KUKA KRL program: Milling_7_33.src

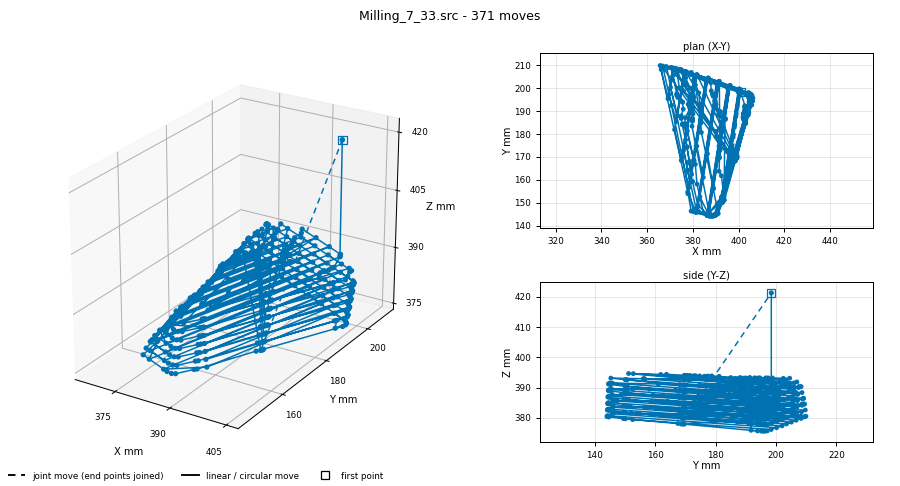
[picture p0: tool path of Milling_7_33.src, 371 of 373 moves have a stored position in this frame; points joined in program order, loops and branches not executed]
&ACCESS RVP
&REL 1
&PARAM TEMPLATE = C:\KRC\Roboter\Template\vorgabe
&PARAM EDITMASK = *
DEF Milling_7_33 ( )


;FOLD INI
;FOLD BASISTECH INI
GLOBAL INTERRUPT DECL 3 WHEN $STOPMESS==TRUE DO IR_STOPM ( )
INTERRUPT ON 3
BAS (#INITMOV,0 )
;ENDFOLD (BASISTECH INI)
;ENDFOLD (INI)

;FOLD STARTPOSITION - BASE IS 0, TOOL IS 5, SPEED IS 15%, POSITION IS A1 5,A2 -90,A3 100,A4 5,A5 -10,A6 -5,E1 0,E2 0,E3 0,E4 0
$BWDSTART = FALSE
PDAT_ACT = {VEL 15,ACC 100,APO_DIST 50}
FDAT_ACT = {TOOL_NO 5,BASE_NO 0,IPO_FRAME #BASE}
BAS (#PTP_PARAMS,15)
PTP  {A1 5,A2 -90,A3 100,A4 5,A5 -10,A6 -5,E1 0,E2 0,E3 0,E4 0}
;ENDFOLD

;FOLD LIN SPEED IS 0.1 m/sec, INTERPOLATION SETTINGS IN FOLD
$VEL.CP=0.1
$ADVANCE=3
;ENDFOLD

BAS(#VEL_PTP,2)
PTP {X 400.878, Y 198.448, Z 421.334, A -161.652, B 81.275, C -141.67, E1 0, E2 0, E3 0, E4 0, S 'B010'}
$VEL.CP=0.012
LIN {X 400.878, Y 198.448, Z 391.334, A -161.652, B 81.275, C -141.67, E1 0, E2 0, E3 0, E4 0}
LIN {X 393.619, Y 152.751, Z 394.599, A -161.652, B 81.275, C -141.67, E1 0, E2 0, E3 0, E4 0}
LIN {X 394.006, Y 186.825, Z 392.897, A -161.652, B 81.275, C -141.67, E1 0, E2 0, E3 0, E4 0}
LIN {X 396.301, Y 201.276, Z 391.864, A -161.652, B 81.275, C -141.67, E1 0, E2 0, E3 0, E4 0}
LIN {X 393.921, Y 186.294, Z 392.935, A -161.652, B 81.275, C -141.67, E1 0, E2 0, E3 0, E4 0}
LIN {X 391.87, Y 173.383, Z 393.857, A -161.652, B 81.275, C -141.67, E1 0, E2 0, E3 0, E4 0}
LIN {X 391.404, Y 170.446, Z 394.067, A -161.652, B 81.275, C -141.67, E1 0, E2 0, E3 0, E4 0}
LIN {X 391.763, Y 172.709, Z 393.905, A -161.652, B 81.275, C -141.67, E1 0, E2 0, E3 0, E4 0}
LIN {X 391.558, Y 203.055, Z 392.469, A -161.652, B 81.275, C -141.67, E1 0, E2 0, E3 0, E4 0}
LIN {X 389.984, Y 193.152, Z 393.177, A -161.652, B 81.275, C -141.67, E1 0, E2 0, E3 0, E4 0}
LIN {X 399.127, Y 169.429, Z 392.991, A -161.652, B 81.275, C -141.67, E1 0, E2 0, E3 0, E4 0}
LIN {X 399.345, Y 169.891, Z 392.937, A -161.652, B 81.275, C -141.67, E1 0, E2 0, E3 0, E4 0}
LIN {X 399.292, Y 170.395, Z 392.92, A -161.652, B 81.275, C -141.67, E1 0, E2 0, E3 0, E4 0}
LIN {X 403.099, Y 184.627, Z 391.678, A -161.652, B 81.275, C -141.67, E1 0, E2 0, E3 0, E4 0}
LIN {X 402.072, Y 186.427, Z 391.741, A -161.652, B 81.275, C -141.67, E1 0, E2 0, E3 0, E4 0}
LIN {X 401.883, Y 187.353, Z 391.724, A -161.652, B 81.275, C -141.67, E1 0, E2 0, E3 0, E4 0}
LIN {X 402.049, Y 188.531, Z 391.643, A -161.652, B 81.275, C -141.67, E1 0, E2 0, E3 0, E4 0}
LIN {X 401.981, Y 188.771, Z 391.641, A -161.652, B 81.275, C -141.67, E1 0, E2 0, E3 0, E4 0}
LIN {X 401.995, Y 188.923, Z 391.631, A -161.652, B 81.275, C -141.67, E1 0, E2 0, E3 0, E4 0}
LIN {X 402.517, Y 190.32, Z 391.488, A -161.652, B 81.275, C -141.67, E1 0, E2 0, E3 0, E4 0}
LIN {X 402.552, Y 191.698, Z 391.416, A -161.652, B 81.275, C -141.67, E1 0, E2 0, E3 0, E4 0}
LIN {X 402.684, Y 192.078, Z 391.379, A -161.652, B 81.275, C -141.67, E1 0, E2 0, E3 0, E4 0}
LIN {X 402.701, Y 192.377, Z 391.362, A -161.652, B 81.275, C -141.67, E1 0, E2 0, E3 0, E4 0}
LIN {X 400.745, Y 198.773, Z 391.338, A -161.652, B 81.275, C -141.67, E1 0, E2 0, E3 0, E4 0}
LIN {X 400.366, Y 199.42, Z 391.362, A -161.652, B 81.275, C -141.67, E1 0, E2 0, E3 0, E4 0}
LIN {X 400.287, Y 199.785, Z 391.355, A -161.652, B 81.275, C -141.67, E1 0, E2 0, E3 0, E4 0}
LIN {X 386.775, Y 204.544, Z 393.094, A -161.652, B 81.275, C -141.67, E1 0, E2 0, E3 0, E4 0}
LIN {X 387.794, Y 202.431, Z 393.048, A -161.652, B 81.275, C -141.67, E1 0, E2 0, E3 0, E4 0}
LIN {X 388.016, Y 198.85, Z 393.188, A -161.652, B 81.275, C -141.67, E1 0, E2 0, E3 0, E4 0}
LIN {X 388.509, Y 197.466, Z 393.183, A -161.652, B 81.275, C -141.67, E1 0, E2 0, E3 0, E4 0}
LIN {X 388.922, Y 196.935, Z 393.149, A -161.652, B 81.275, C -141.67, E1 0, E2 0, E3 0, E4 0}
LIN {X 388.831, Y 196.544, Z 393.181, A -161.652, B 81.275, C -141.67, E1 0, E2 0, E3 0, E4 0}
LIN {X 389.518, Y 194.72, Z 393.169, A -161.652, B 81.275, C -141.67, E1 0, E2 0, E3 0, E4 0}
LIN {X 389.72, Y 194.484, Z 393.151, A -161.652, B 81.275, C -141.67, E1 0, E2 0, E3 0, E4 0}
LIN {X 389.694, Y 194.079, Z 393.174, A -161.652, B 81.275, C -141.67, E1 0, E2 0, E3 0, E4 0}
LIN {X 390.083, Y 192.837, Z 393.178, A -161.652, B 81.275, C -141.67, E1 0, E2 0, E3 0, E4 0}
LIN {X 389.807, Y 191.398, Z 393.287, A -161.652, B 81.275, C -141.67, E1 0, E2 0, E3 0, E4 0}
LIN {X 390.122, Y 191.272, Z 393.247, A -161.652, B 81.275, C -141.67, E1 0, E2 0, E3 0, E4 0}
LIN {X 391.067, Y 190.153, Z 393.164, A -161.652, B 81.275, C -141.67, E1 0, E2 0, E3 0, E4 0}
LIN {X 392.007, Y 189.84, Z 393.042, A -161.652, B 81.275, C -141.67, E1 0, E2 0, E3 0, E4 0}
LIN {X 391.95, Y 189.635, Z 393.06, A -161.652, B 81.275, C -141.67, E1 0, E2 0, E3 0, E4 0}
LIN {X 391.422, Y 189.417, Z 393.148, A -161.652, B 81.275, C -141.67, E1 0, E2 0, E3 0, E4 0}
LIN {X 391.115, Y 188.334, Z 393.245, A -161.652, B 81.275, C -141.67, E1 0, E2 0, E3 0, E4 0}
LIN {X 391.663, Y 187.948, Z 393.184, A -161.652, B 81.275, C -141.67, E1 0, E2 0, E3 0, E4 0}
LIN {X 391.707, Y 187.877, Z 393.181, A -161.652, B 81.275, C -141.67, E1 0, E2 0, E3 0, E4 0}
LIN {X 394.151, Y 186.717, Z 392.881, A -161.652, B 81.275, C -141.67, E1 0, E2 0, E3 0, E4 0}
LIN {X 394.211, Y 186.575, Z 392.879, A -161.652, B 81.275, C -141.67, E1 0, E2 0, E3 0, E4 0}
LIN {X 394.18, Y 186.468, Z 392.889, A -161.652, B 81.275, C -141.67, E1 0, E2 0, E3 0, E4 0}
LIN {X 392.665, Y 185.296, Z 393.166, A -161.652, B 81.275, C -141.67, E1 0, E2 0, E3 0, E4 0}
LIN {X 392.584, Y 185.05, Z 393.189, A -161.652, B 81.275, C -141.67, E1 0, E2 0, E3 0, E4 0}
LIN {X 392.401, Y 184.875, Z 393.225, A -161.652, B 81.275, C -141.67, E1 0, E2 0, E3 0, E4 0}
LIN {X 390.283, Y 181.178, Z 393.712, A -161.652, B 81.275, C -141.67, E1 0, E2 0, E3 0, E4 0}
LIN {X 390.068, Y 178.729, Z 393.861, A -161.652, B 81.275, C -141.67, E1 0, E2 0, E3 0, E4 0}
LIN {X 390.889, Y 177.56, Z 393.798, A -161.652, B 81.275, C -141.67, E1 0, E2 0, E3 0, E4 0}
LIN {X 391.421, Y 177.182, Z 393.739, A -161.652, B 81.275, C -141.67, E1 0, E2 0, E3 0, E4 0}
LIN {X 391.585, Y 176.323, Z 393.757, A -161.652, B 81.275, C -141.67, E1 0, E2 0, E3 0, E4 0}
LIN {X 391.395, Y 174.71, Z 393.862, A -161.652, B 81.275, C -141.67, E1 0, E2 0, E3 0, E4 0}
LIN {X 391.897, Y 173.324, Z 393.856, A -161.652, B 81.275, C -141.67, E1 0, E2 0, E3 0, E4 0}
LIN {X 391.285, Y 171.448, Z 394.036, A -161.652, B 81.275, C -141.67, E1 0, E2 0, E3 0, E4 0}
LIN {X 391.647, Y 169.624, Z 394.071, A -161.652, B 81.275, C -141.67, E1 0, E2 0, E3 0, E4 0}
LIN {X 391.444, Y 163.743, Z 394.385, A -161.652, B 81.275, C -141.67, E1 0, E2 0, E3 0, E4 0}
LIN {X 392.448, Y 161.811, Z 394.332, A -161.652, B 81.275, C -141.67, E1 0, E2 0, E3 0, E4 0}
LIN {X 393.769, Y 151.184, Z 394.653, A -161.652, B 81.275, C -141.67, E1 0, E2 0, E3 0, E4 0}
LIN {X 398.578, Y 168.267, Z 393.127, A -161.652, B 81.275, C -141.67, E1 0, E2 0, E3 0, E4 0}
LIN {X 399.127, Y 169.429, Z 392.991, A -161.652, B 81.275, C -141.67, E1 0, E2 0, E3 0, E4 0}
LIN {X 405.47, Y 194.853, Z 390.839, A -161.652, B 81.275, C -141.67, E1 0, E2 0, E3 0, E4 0}
LIN {X 405.157, Y 194.749, Z 388.69, A -161.652, B 81.275, C -141.67, E1 0, E2 0, E3 0, E4 0}
LIN {X 404.147, Y 188.389, Z 389.144, A -161.652, B 81.275, C -141.67, E1 0, E2 0, E3 0, E4 0}
LIN {X 404.127, Y 188.266, Z 389.153, A -161.652, B 81.275, C -141.67, E1 0, E2 0, E3 0, E4 0}
LIN {X 393.098, Y 150.478, Z 392.585, A -161.652, B 81.275, C -141.67, E1 0, E2 0, E3 0, E4 0}
LIN {X 400.861, Y 199.348, Z 389.094, A -161.652, B 81.275, C -141.67, E1 0, E2 0, E3 0, E4 0}
LIN {X 396.117, Y 201.124, Z 389.699, A -161.652, B 81.275, C -141.67, E1 0, E2 0, E3 0, E4 0}
LIN {X 388.958, Y 156.06, Z 392.919, A -161.652, B 81.275, C -141.67, E1 0, E2 0, E3 0, E4 0}
LIN {X 386.363, Y 171.36, Z 392.558, A -161.652, B 81.275, C -141.67, E1 0, E2 0, E3 0, E4 0}
LIN {X 391.374, Y 202.909, Z 390.304, A -161.652, B 81.275, C -141.67, E1 0, E2 0, E3 0, E4 0}
LIN {X 386.584, Y 204.395, Z 390.93, A -161.652, B 81.275, C -141.67, E1 0, E2 0, E3 0, E4 0}
LIN {X 383.47, Y 184.793, Z 392.33, A -161.652, B 81.275, C -141.67, E1 0, E2 0, E3 0, E4 0}
LIN {X 381.086, Y 201.427, Z 391.874, A -161.652, B 81.275, C -141.67, E1 0, E2 0, E3 0, E4 0}
LIN {X 381.812, Y 205.993, Z 391.547, A -161.652, B 81.275, C -141.67, E1 0, E2 0, E3 0, E4 0}
LIN {X 398.814, Y 169.325, Z 390.842, A -161.652, B 81.275, C -141.67, E1 0, E2 0, E3 0, E4 0}
LIN {X 399.032, Y 169.787, Z 390.788, A -161.652, B 81.275, C -141.67, E1 0, E2 0, E3 0, E4 0}
LIN {X 398.979, Y 170.292, Z 390.772, A -161.652, B 81.275, C -141.67, E1 0, E2 0, E3 0, E4 0}
LIN {X 405.704, Y 192.648, Z 388.712, A -161.652, B 81.275, C -141.67, E1 0, E2 0, E3 0, E4 0}
LIN {X 404.345, Y 197.182, Z 388.691, A -161.652, B 81.275, C -141.67, E1 0, E2 0, E3 0, E4 0}
LIN {X 404.324, Y 198.143, Z 388.647, A -161.652, B 81.275, C -141.67, E1 0, E2 0, E3 0, E4 0}
LIN {X 379.268, Y 206.924, Z 391.873, A -161.652, B 81.275, C -141.67, E1 0, E2 0, E3 0, E4 0}
LIN {X 380.336, Y 203.608, Z 391.878, A -161.652, B 81.275, C -141.67, E1 0, E2 0, E3 0, E4 0}
LIN {X 380.622, Y 203.285, Z 391.852, A -161.652, B 81.275, C -141.67, E1 0, E2 0, E3 0, E4 0}
LIN {X 382.552, Y 198.008, Z 391.825, A -161.652, B 81.275, C -141.67, E1 0, E2 0, E3 0, E4 0}
LIN {X 383.125, Y 193.065, Z 391.981, A -161.652, B 81.275, C -141.67, E1 0, E2 0, E3 0, E4 0}
LIN {X 383.514, Y 192.671, Z 391.943, A -161.652, B 81.275, C -141.67, E1 0, E2 0, E3 0, E4 0}
LIN {X 383.065, Y 191.799, Z 392.051, A -161.652, B 81.275, C -141.67, E1 0, E2 0, E3 0, E4 0}
LIN {X 382.999, Y 190.748, Z 392.111, A -161.652, B 81.275, C -141.67, E1 0, E2 0, E3 0, E4 0}
LIN {X 383.489, Y 190.213, Z 392.065, A -161.652, B 81.275, C -141.67, E1 0, E2 0, E3 0, E4 0}
LIN {X 383.697, Y 189.753, Z 392.057, A -161.652, B 81.275, C -141.67, E1 0, E2 0, E3 0, E4 0}
LIN {X 383.834, Y 187.857, Z 392.129, A -161.652, B 81.275, C -141.67, E1 0, E2 0, E3 0, E4 0}
LIN {X 383.324, Y 186.499, Z 392.269, A -161.652, B 81.275, C -141.67, E1 0, E2 0, E3 0, E4 0}
LIN {X 383.699, Y 180.729, Z 392.493, A -161.652, B 81.275, C -141.67, E1 0, E2 0, E3 0, E4 0}
LIN {X 388.902, Y 156.463, Z 392.908, A -161.652, B 81.275, C -141.67, E1 0, E2 0, E3 0, E4 0}
LIN {X 388.849, Y 156.343, Z 392.921, A -161.652, B 81.275, C -141.67, E1 0, E2 0, E3 0, E4 0}
LIN {X 391.072, Y 145.307, Z 393.13, A -161.652, B 81.275, C -141.67, E1 0, E2 0, E3 0, E4 0}
LIN {X 392.895, Y 150.059, Z 392.635, A -161.652, B 81.275, C -141.67, E1 0, E2 0, E3 0, E4 0}
LIN {X 393.255, Y 150.719, Z 392.551, A -161.652, B 81.275, C -141.67, E1 0, E2 0, E3 0, E4 0}
LIN {X 398.265, Y 168.163, Z 390.978, A -161.652, B 81.275, C -141.67, E1 0, E2 0, E3 0, E4 0}
LIN {X 398.814, Y 169.325, Z 390.842, A -161.652, B 81.275, C -141.67, E1 0, E2 0, E3 0, E4 0}
LIN {X 404.432, Y 189.322, Z 389.058, A -161.652, B 81.275, C -141.67, E1 0, E2 0, E3 0, E4 0}
LIN {X 404.119, Y 189.218, Z 386.909, A -161.652, B 81.275, C -141.67, E1 0, E2 0, E3 0, E4 0}
LIN {X 405.395, Y 197.252, Z 386.335, A -161.652, B 81.275, C -141.67, E1 0, E2 0, E3 0, E4 0}
LIN {X 400.677, Y 199.196, Z 386.928, A -161.652, B 81.275, C -141.67, E1 0, E2 0, E3 0, E4 0}
LIN {X 392.967, Y 150.66, Z 390.396, A -161.652, B 81.275, C -141.67, E1 0, E2 0, E3 0, E4 0}
LIN {X 387.172, Y 145.821, Z 391.474, A -161.652, B 81.275, C -141.67, E1 0, E2 0, E3 0, E4 0}
LIN {X 395.933, Y 200.972, Z 387.534, A -161.652, B 81.275, C -141.67, E1 0, E2 0, E3 0, E4 0}
LIN {X 391.191, Y 202.763, Z 388.138, A -161.652, B 81.275, C -141.67, E1 0, E2 0, E3 0, E4 0}
LIN {X 384.565, Y 161.049, Z 391.118, A -161.652, B 81.275, C -141.67, E1 0, E2 0, E3 0, E4 0}
LIN {X 381.709, Y 174.714, Z 390.874, A -161.652, B 81.275, C -141.67, E1 0, E2 0, E3 0, E4 0}
LIN {X 386.4, Y 204.243, Z 388.764, A -161.652, B 81.275, C -141.67, E1 0, E2 0, E3 0, E4 0}
LIN {X 381.628, Y 205.845, Z 389.382, A -161.652, B 81.275, C -141.67, E1 0, E2 0, E3 0, E4 0}
LIN {X 380.214, Y 196.943, Z 390.018, A -161.652, B 81.275, C -141.67, E1 0, E2 0, E3 0, E4 0}
LIN {X 376.502, Y 205.217, Z 390.159, A -161.652, B 81.275, C -141.67, E1 0, E2 0, E3 0, E4 0}
LIN {X 376.853, Y 207.424, Z 390.001, A -161.652, B 81.275, C -141.67, E1 0, E2 0, E3 0, E4 0}
LIN {X 398.501, Y 169.221, Z 388.694, A -161.652, B 81.275, C -141.67, E1 0, E2 0, E3 0, E4 0}
LIN {X 398.719, Y 169.683, Z 388.639, A -161.652, B 81.275, C -141.67, E1 0, E2 0, E3 0, E4 0}
LIN {X 398.666, Y 170.188, Z 388.623, A -161.652, B 81.275, C -141.67, E1 0, E2 0, E3 0, E4 0}
LIN {X 406.112, Y 194.409, Z 386.368, A -161.652, B 81.275, C -141.67, E1 0, E2 0, E3 0, E4 0}
LIN {X 406.209, Y 195.704, Z 386.291, A -161.652, B 81.275, C -141.67, E1 0, E2 0, E3 0, E4 0}
LIN {X 405.842, Y 196.798, Z 386.292, A -161.652, B 81.275, C -141.67, E1 0, E2 0, E3 0, E4 0}
LIN {X 405.035, Y 197.632, Z 386.369, A -161.652, B 81.275, C -141.67, E1 0, E2 0, E3 0, E4 0}
LIN {X 375.02, Y 208.084, Z 390.236, A -161.652, B 81.275, C -141.67, E1 0, E2 0, E3 0, E4 0}
LIN {X 374.358, Y 208.308, Z 390.322, A -161.652, B 81.275, C -141.67, E1 0, E2 0, E3 0, E4 0}
LIN {X 374.534, Y 207.575, Z 390.332, A -161.652, B 81.275, C -141.67, E1 0, E2 0, E3 0, E4 0}
LIN {X 376.096, Y 206.013, Z 390.18, A -161.652, B 81.275, C -141.67, E1 0, E2 0, E3 0, E4 0}
LIN {X 376.852, Y 204.524, Z 390.142, A -161.652, B 81.275, C -141.67, E1 0, E2 0, E3 0, E4 0}
LIN {X 376.834, Y 202.424, Z 390.246, A -161.652, B 81.275, C -141.67, E1 0, E2 0, E3 0, E4 0}
LIN {X 377.215, Y 201.348, Z 390.242, A -161.652, B 81.275, C -141.67, E1 0, E2 0, E3 0, E4 0}
LIN {X 378.866, Y 200.125, Z 390.061, A -161.652, B 81.275, C -141.67, E1 0, E2 0, E3 0, E4 0}
LIN {X 380.483, Y 195.935, Z 390.028, A -161.652, B 81.275, C -141.67, E1 0, E2 0, E3 0, E4 0}
LIN {X 380.186, Y 191.634, Z 390.279, A -161.652, B 81.275, C -141.67, E1 0, E2 0, E3 0, E4 0}
LIN {X 379.523, Y 190.108, Z 390.449, A -161.652, B 81.275, C -141.67, E1 0, E2 0, E3 0, E4 0}
LIN {X 379.535, Y 189.929, Z 390.456, A -161.652, B 81.275, C -141.67, E1 0, E2 0, E3 0, E4 0}
LIN {X 380.044, Y 188.758, Z 390.438, A -161.652, B 81.275, C -141.67, E1 0, E2 0, E3 0, E4 0}
LIN {X 379.694, Y 186.845, Z 390.582, A -161.652, B 81.275, C -141.67, E1 0, E2 0, E3 0, E4 0}
LIN {X 379.936, Y 186.659, Z 390.555, A -161.652, B 81.275, C -141.67, E1 0, E2 0, E3 0, E4 0}
LIN {X 379.822, Y 185.764, Z 390.615, A -161.652, B 81.275, C -141.67, E1 0, E2 0, E3 0, E4 0}
LIN {X 379.75, Y 185.636, Z 390.632, A -161.652, B 81.275, C -141.67, E1 0, E2 0, E3 0, E4 0}
LIN {X 379.596, Y 183.433, Z 390.761, A -161.652, B 81.275, C -141.67, E1 0, E2 0, E3 0, E4 0}
LIN {X 387.223, Y 144.971, Z 391.508, A -161.652, B 81.275, C -141.67, E1 0, E2 0, E3 0, E4 0}
LIN {X 388.845, Y 144.572, Z 391.291, A -161.652, B 81.275, C -141.67, E1 0, E2 0, E3 0, E4 0}
LIN {X 390.047, Y 144.577, Z 391.116, A -161.652, B 81.275, C -141.67, E1 0, E2 0, E3 0, E4 0}
LIN {X 390.749, Y 145.187, Z 390.984, A -161.652, B 81.275, C -141.67, E1 0, E2 0, E3 0, E4 0}
LIN {X 392.582, Y 149.956, Z 390.487, A -161.652, B 81.275, C -141.67, E1 0, E2 0, E3 0, E4 0}
LIN {X 392.943, Y 150.616, Z 390.402, A -161.652, B 81.275, C -141.67, E1 0, E2 0, E3 0, E4 0}
LIN {X 397.952, Y 168.06, Z 388.83, A -161.652, B 81.275, C -141.67, E1 0, E2 0, E3 0, E4 0}
LIN {X 398.501, Y 169.221, Z 388.694, A -161.652, B 81.275, C -141.67, E1 0, E2 0, E3 0, E4 0}
LIN {X 405.512, Y 197.128, Z 386.324, A -161.652, B 81.275, C -141.67, E1 0, E2 0, E3 0, E4 0}
LIN {X 405.199, Y 197.024, Z 384.175, A -161.652, B 81.275, C -141.67, E1 0, E2 0, E3 0, E4 0}
LIN {X 404.057, Y 189.835, Z 384.689, A -161.652, B 81.275, C -141.67, E1 0, E2 0, E3 0, E4 0}
LIN {X 392.845, Y 150.9, Z 388.203, A -161.652, B 81.275, C -141.67, E1 0, E2 0, E3 0, E4 0}
LIN {X 400.493, Y 199.044, Z 384.763, A -161.652, B 81.275, C -141.67, E1 0, E2 0, E3 0, E4 0}
LIN {X 395.749, Y 200.821, Z 385.368, A -161.652, B 81.275, C -141.67, E1 0, E2 0, E3 0, E4 0}
LIN {X 386.862, Y 144.877, Z 389.366, A -161.652, B 81.275, C -141.67, E1 0, E2 0, E3 0, E4 0}
LIN {X 383.063, Y 152.603, Z 389.546, A -161.652, B 81.275, C -141.67, E1 0, E2 0, E3 0, E4 0}
LIN {X 391.008, Y 202.617, Z 385.972, A -161.652, B 81.275, C -141.67, E1 0, E2 0, E3 0, E4 0}
LIN {X 386.216, Y 204.09, Z 386.599, A -161.652, B 81.275, C -141.67, E1 0, E2 0, E3 0, E4 0}
LIN {X 380.518, Y 168.22, Z 389.162, A -161.652, B 81.275, C -141.67, E1 0, E2 0, E3 0, E4 0}
LIN {X 377.579, Y 181.361, Z 388.955, A -161.652, B 81.275, C -141.67, E1 0, E2 0, E3 0, E4 0}
LIN {X 381.445, Y 205.697, Z 387.216, A -161.652, B 81.275, C -141.67, E1 0, E2 0, E3 0, E4 0}
LIN {X 376.669, Y 207.274, Z 387.836, A -161.652, B 81.275, C -141.67, E1 0, E2 0, E3 0, E4 0}
LIN {X 375.369, Y 199.091, Z 388.421, A -161.652, B 81.275, C -141.67, E1 0, E2 0, E3 0, E4 0}
LIN {X 398.187, Y 169.117, Z 386.545, A -161.652, B 81.275, C -141.67, E1 0, E2 0, E3 0, E4 0}
LIN {X 398.406, Y 169.579, Z 386.491, A -161.652, B 81.275, C -141.67, E1 0, E2 0, E3 0, E4 0}
LIN {X 398.353, Y 170.084, Z 386.474, A -161.652, B 81.275, C -141.67, E1 0, E2 0, E3 0, E4 0}
LIN {X 405.799, Y 194.306, Z 384.219, A -161.652, B 81.275, C -141.67, E1 0, E2 0, E3 0, E4 0}
LIN {X 405.896, Y 195.6, Z 384.143, A -161.652, B 81.275, C -141.67, E1 0, E2 0, E3 0, E4 0}
LIN {X 405.529, Y 196.694, Z 384.143, A -161.652, B 81.275, C -141.67, E1 0, E2 0, E3 0, E4 0}
LIN {X 404.722, Y 197.529, Z 384.22, A -161.652, B 81.275, C -141.67, E1 0, E2 0, E3 0, E4 0}
LIN {X 377.455, Y 206.991, Z 387.735, A -161.652, B 81.275, C -141.67, E1 0, E2 0, E3 0, E4 0}
LIN {X 372.794, Y 208.629, Z 388.335, A -161.652, B 81.275, C -141.67, E1 0, E2 0, E3 0, E4 0}
LIN {X 372.835, Y 206.487, Z 388.433, A -161.652, B 81.275, C -141.67, E1 0, E2 0, E3 0, E4 0}
LIN {X 373.226, Y 205.815, Z 388.408, A -161.652, B 81.275, C -141.67, E1 0, E2 0, E3 0, E4 0}
LIN {X 374.071, Y 200.184, Z 388.557, A -161.652, B 81.275, C -141.67, E1 0, E2 0, E3 0, E4 0}
LIN {X 375.592, Y 198.876, Z 388.399, A -161.652, B 81.275, C -141.67, E1 0, E2 0, E3 0, E4 0}
LIN {X 375.921, Y 198.764, Z 388.356, A -161.652, B 81.275, C -141.67, E1 0, E2 0, E3 0, E4 0}
LIN {X 378.592, Y 196.44, Z 388.079, A -161.652, B 81.275, C -141.67, E1 0, E2 0, E3 0, E4 0}
LIN {X 378.73, Y 195.153, Z 388.121, A -161.652, B 81.275, C -141.67, E1 0, E2 0, E3 0, E4 0}
LIN {X 378.823, Y 194.956, Z 388.117, A -161.652, B 81.275, C -141.67, E1 0, E2 0, E3 0, E4 0}
LIN {X 378.747, Y 194.903, Z 388.131, A -161.652, B 81.275, C -141.67, E1 0, E2 0, E3 0, E4 0}
LIN {X 377.933, Y 193.083, Z 388.337, A -161.652, B 81.275, C -141.67, E1 0, E2 0, E3 0, E4 0}
LIN {X 378.01, Y 192.879, Z 388.336, A -161.652, B 81.275, C -141.67, E1 0, E2 0, E3 0, E4 0}
LIN {X 378.323, Y 192.721, Z 388.298, A -161.652, B 81.275, C -141.67, E1 0, E2 0, E3 0, E4 0}
LIN {X 378.555, Y 191.71, Z 388.313, A -161.652, B 81.275, C -141.67, E1 0, E2 0, E3 0, E4 0}
LIN {X 378.753, Y 191.206, Z 388.309, A -161.652, B 81.275, C -141.67, E1 0, E2 0, E3 0, E4 0}
LIN {X 376.678, Y 187.15, Z 388.807, A -161.652, B 81.275, C -141.67, E1 0, E2 0, E3 0, E4 0}
LIN {X 376.488, Y 184.579, Z 388.959, A -161.652, B 81.275, C -141.67, E1 0, E2 0, E3 0, E4 0}
LIN {X 376.688, Y 183.18, Z 388.997, A -161.652, B 81.275, C -141.67, E1 0, E2 0, E3 0, E4 0}
LIN {X 377.282, Y 181.96, Z 388.97, A -161.652, B 81.275, C -141.67, E1 0, E2 0, E3 0, E4 0}
LIN {X 380.4, Y 168.673, Z 389.157, A -161.652, B 81.275, C -141.67, E1 0, E2 0, E3 0, E4 0}
LIN {X 380.38, Y 168.592, Z 389.164, A -161.652, B 81.275, C -141.67, E1 0, E2 0, E3 0, E4 0}
LIN {X 381.071, Y 166.766, Z 389.152, A -161.652, B 81.275, C -141.67, E1 0, E2 0, E3 0, E4 0}
LIN {X 381.789, Y 158.113, Z 389.465, A -161.652, B 81.275, C -141.67, E1 0, E2 0, E3 0, E4 0}
LIN {X 384.674, Y 145.451, Z 389.657, A -161.652, B 81.275, C -141.67, E1 0, E2 0, E3 0, E4 0}
LIN {X 388.532, Y 144.468, Z 389.142, A -161.652, B 81.275, C -141.67, E1 0, E2 0, E3 0, E4 0}
LIN {X 389.734, Y 144.473, Z 388.967, A -161.652, B 81.275, C -141.67, E1 0, E2 0, E3 0, E4 0}
LIN {X 390.436, Y 145.083, Z 388.835, A -161.652, B 81.275, C -141.67, E1 0, E2 0, E3 0, E4 0}
LIN {X 392.269, Y 149.852, Z 388.338, A -161.652, B 81.275, C -141.67, E1 0, E2 0, E3 0, E4 0}
LIN {X 392.63, Y 150.512, Z 388.253, A -161.652, B 81.275, C -141.67, E1 0, E2 0, E3 0, E4 0}
LIN {X 397.639, Y 167.956, Z 386.681, A -161.652, B 81.275, C -141.67, E1 0, E2 0, E3 0, E4 0}
LIN {X 398.187, Y 169.117, Z 386.545, A -161.652, B 81.275, C -141.67, E1 0, E2 0, E3 0, E4 0}
LIN {X 405.316, Y 196.902, Z 384.164, A -161.652, B 81.275, C -141.67, E1 0, E2 0, E3 0, E4 0}
LIN {X 405.003, Y 196.798, Z 382.015, A -161.652, B 81.275, C -141.67, E1 0, E2 0, E3 0, E4 0}
LIN {X 403.964, Y 190.258, Z 382.483, A -161.652, B 81.275, C -141.67, E1 0, E2 0, E3 0, E4 0}
LIN {X 392.737, Y 151.225, Z 386.004, A -161.652, B 81.275, C -141.67, E1 0, E2 0, E3 0, E4 0}
LIN {X 400.309, Y 198.891, Z 382.598, A -161.652, B 81.275, C -141.67, E1 0, E2 0, E3 0, E4 0}
LIN {X 395.565, Y 200.669, Z 383.203, A -161.652, B 81.275, C -141.67, E1 0, E2 0, E3 0, E4 0}
LIN {X 386.681, Y 144.746, Z 387.199, A -161.652, B 81.275, C -141.67, E1 0, E2 0, E3 0, E4 0}
LIN {X 382.288, Y 148.728, Z 387.647, A -161.652, B 81.275, C -141.67, E1 0, E2 0, E3 0, E4 0}
LIN {X 390.825, Y 202.471, Z 383.807, A -161.652, B 81.275, C -141.67, E1 0, E2 0, E3 0, E4 0}
LIN {X 386.032, Y 203.938, Z 384.434, A -161.652, B 81.275, C -141.67, E1 0, E2 0, E3 0, E4 0}
LIN {X 379.432, Y 162.392, Z 387.403, A -161.652, B 81.275, C -141.67, E1 0, E2 0, E3 0, E4 0}
LIN {X 376.803, Y 177.484, Z 387.056, A -161.652, B 81.275, C -141.67, E1 0, E2 0, E3 0, E4 0}
LIN {X 381.261, Y 205.549, Z 385.051, A -161.652, B 81.275, C -141.67, E1 0, E2 0, E3 0, E4 0}
LIN {X 376.485, Y 207.124, Z 385.671, A -161.652, B 81.275, C -141.67, E1 0, E2 0, E3 0, E4 0}
LIN {X 374.541, Y 194.887, Z 386.545, A -161.652, B 81.275, C -141.67, E1 0, E2 0, E3 0, E4 0}
LIN {X 371.186, Y 205.406, Z 386.526, A -161.652, B 81.275, C -141.67, E1 0, E2 0, E3 0, E4 0}
LIN {X 371.722, Y 208.782, Z 386.284, A -161.652, B 81.275, C -141.67, E1 0, E2 0, E3 0, E4 0}
LIN {X 397.874, Y 169.013, Z 384.396, A -161.652, B 81.275, C -141.67, E1 0, E2 0, E3 0, E4 0}
LIN {X 398.093, Y 169.476, Z 384.342, A -161.652, B 81.275, C -141.67, E1 0, E2 0, E3 0, E4 0}
LIN {X 398.04, Y 169.98, Z 384.325, A -161.652, B 81.275, C -141.67, E1 0, E2 0, E3 0, E4 0}
LIN {X 405.486, Y 194.202, Z 382.07, A -161.652, B 81.275, C -141.67, E1 0, E2 0, E3 0, E4 0}
LIN {X 405.583, Y 195.496, Z 381.994, A -161.652, B 81.275, C -141.67, E1 0, E2 0, E3 0, E4 0}
LIN {X 405.216, Y 196.59, Z 381.994, A -161.652, B 81.275, C -141.67, E1 0, E2 0, E3 0, E4 0}
LIN {X 404.409, Y 197.425, Z 382.071, A -161.652, B 81.275, C -141.67, E1 0, E2 0, E3 0, E4 0}
LIN {X 370.573, Y 209.12, Z 386.435, A -161.652, B 81.275, C -141.67, E1 0, E2 0, E3 0, E4 0}
LIN {X 370.483, Y 209.139, Z 386.448, A -161.652, B 81.275, C -141.67, E1 0, E2 0, E3 0, E4 0}
LIN {X 372.917, Y 197.66, Z 386.648, A -161.652, B 81.275, C -141.67, E1 0, E2 0, E3 0, E4 0}
LIN {X 372.91, Y 197.002, Z 386.68, A -161.652, B 81.275, C -141.67, E1 0, E2 0, E3 0, E4 0}
LIN {X 373.373, Y 195.981, Z 386.662, A -161.652, B 81.275, C -141.67, E1 0, E2 0, E3 0, E4 0}
LIN {X 375.465, Y 193.981, Z 386.454, A -161.652, B 81.275, C -141.67, E1 0, E2 0, E3 0, E4 0}
LIN {X 375.494, Y 193.912, Z 386.453, A -161.652, B 81.275, C -141.67, E1 0, E2 0, E3 0, E4 0}
LIN {X 375.783, Y 190.907, Z 386.556, A -161.652, B 81.275, C -141.67, E1 0, E2 0, E3 0, E4 0}
LIN {X 374.895, Y 187.953, Z 386.828, A -161.652, B 81.275, C -141.67, E1 0, E2 0, E3 0, E4 0}
LIN {X 374.859, Y 186.824, Z 386.888, A -161.652, B 81.275, C -141.67, E1 0, E2 0, E3 0, E4 0}
LIN {X 375.395, Y 184.384, Z 386.928, A -161.652, B 81.275, C -141.67, E1 0, E2 0, E3 0, E4 0}
LIN {X 375.34, Y 184.144, Z 386.948, A -161.652, B 81.275, C -141.67, E1 0, E2 0, E3 0, E4 0}
LIN {X 377.512, Y 174.413, Z 387.102, A -161.652, B 81.275, C -141.67, E1 0, E2 0, E3 0, E4 0}
LIN {X 377.467, Y 174.218, Z 387.118, A -161.652, B 81.275, C -141.67, E1 0, E2 0, E3 0, E4 0}
LIN {X 378.461, Y 168.07, Z 387.27, A -161.652, B 81.275, C -141.67, E1 0, E2 0, E3 0, E4 0}
LIN {X 378.387, Y 167.29, Z 387.318, A -161.652, B 81.275, C -141.67, E1 0, E2 0, E3 0, E4 0}
LIN {X 379.751, Y 159.33, Z 387.504, A -161.652, B 81.275, C -141.67, E1 0, E2 0, E3 0, E4 0}
LIN {X 379.828, Y 159.215, Z 387.498, A -161.652, B 81.275, C -141.67, E1 0, E2 0, E3 0, E4 0}
LIN {X 382.898, Y 145.805, Z 387.699, A -161.652, B 81.275, C -141.67, E1 0, E2 0, E3 0, E4 0}
LIN {X 388.219, Y 144.364, Z 386.993, A -161.652, B 81.275, C -141.67, E1 0, E2 0, E3 0, E4 0}
LIN {X 389.421, Y 144.369, Z 386.818, A -161.652, B 81.275, C -141.67, E1 0, E2 0, E3 0, E4 0}
LIN {X 390.123, Y 144.979, Z 386.686, A -161.652, B 81.275, C -141.67, E1 0, E2 0, E3 0, E4 0}
LIN {X 391.956, Y 149.748, Z 386.189, A -161.652, B 81.275, C -141.67, E1 0, E2 0, E3 0, E4 0}
LIN {X 392.316, Y 150.408, Z 386.105, A -161.652, B 81.275, C -141.67, E1 0, E2 0, E3 0, E4 0}
LIN {X 397.326, Y 167.852, Z 384.532, A -161.652, B 81.275, C -141.67, E1 0, E2 0, E3 0, E4 0}
LIN {X 397.874, Y 169.013, Z 384.396, A -161.652, B 81.275, C -141.67, E1 0, E2 0, E3 0, E4 0}
LIN {X 405.121, Y 196.683, Z 382.004, A -161.652, B 81.275, C -141.67, E1 0, E2 0, E3 0, E4 0}
LIN {X 404.808, Y 196.579, Z 379.855, A -161.652, B 81.275, C -141.67, E1 0, E2 0, E3 0, E4 0}
LIN {X 403.867, Y 190.656, Z 380.278, A -161.652, B 81.275, C -141.67, E1 0, E2 0, E3 0, E4 0}
LIN {X 392.641, Y 151.627, Z 383.799, A -161.652, B 81.275, C -141.67, E1 0, E2 0, E3 0, E4 0}
LIN {X 400.124, Y 198.731, Z 380.433, A -161.652, B 81.275, C -141.67, E1 0, E2 0, E3 0, E4 0}
LIN {X 395.381, Y 200.517, Z 381.038, A -161.652, B 81.275, C -141.67, E1 0, E2 0, E3 0, E4 0}
LIN {X 386.501, Y 144.615, Z 385.032, A -161.652, B 81.275, C -141.67, E1 0, E2 0, E3 0, E4 0}
LIN {X 381.697, Y 146.016, Z 385.664, A -161.652, B 81.275, C -141.67, E1 0, E2 0, E3 0, E4 0}
LIN {X 390.642, Y 202.325, Z 381.641, A -161.652, B 81.275, C -141.67, E1 0, E2 0, E3 0, E4 0}
LIN {X 385.848, Y 203.786, Z 382.269, A -161.652, B 81.275, C -141.67, E1 0, E2 0, E3 0, E4 0}
LIN {X 378.702, Y 158.805, Z 385.483, A -161.652, B 81.275, C -141.67, E1 0, E2 0, E3 0, E4 0}
LIN {X 375.919, Y 172.927, Z 385.206, A -161.652, B 81.275, C -141.67, E1 0, E2 0, E3 0, E4 0}
LIN {X 381.078, Y 205.401, Z 382.885, A -161.652, B 81.275, C -141.67, E1 0, E2 0, E3 0, E4 0}
LIN {X 376.301, Y 206.973, Z 383.505, A -161.652, B 81.275, C -141.67, E1 0, E2 0, E3 0, E4 0}
LIN {X 373.283, Y 187.973, Z 384.863, A -161.652, B 81.275, C -141.67, E1 0, E2 0, E3 0, E4 0}
LIN {X 370.228, Y 200.385, Z 384.708, A -161.652, B 81.275, C -141.67, E1 0, E2 0, E3 0, E4 0}
LIN {X 371.539, Y 208.634, Z 384.119, A -161.652, B 81.275, C -141.67, E1 0, E2 0, E3 0, E4 0}
LIN {X 397.561, Y 168.909, Z 382.247, A -161.652, B 81.275, C -141.67, E1 0, E2 0, E3 0, E4 0}
LIN {X 397.78, Y 169.372, Z 382.193, A -161.652, B 81.275, C -141.67, E1 0, E2 0, E3 0, E4 0}
LIN {X 397.727, Y 169.877, Z 382.177, A -161.652, B 81.275, C -141.67, E1 0, E2 0, E3 0, E4 0}
LIN {X 405.173, Y 194.098, Z 379.921, A -161.652, B 81.275, C -141.67, E1 0, E2 0, E3 0, E4 0}
LIN {X 405.27, Y 195.393, Z 379.845, A -161.652, B 81.275, C -141.67, E1 0, E2 0, E3 0, E4 0}
LIN {X 404.903, Y 196.487, Z 379.845, A -161.652, B 81.275, C -141.67, E1 0, E2 0, E3 0, E4 0}
LIN {X 404.096, Y 197.321, Z 379.923, A -161.652, B 81.275, C -141.67, E1 0, E2 0, E3 0, E4 0}
LIN {X 368.45, Y 209.412, Z 384.531, A -161.652, B 81.275, C -141.67, E1 0, E2 0, E3 0, E4 0}
LIN {X 368.352, Y 209.431, Z 384.545, A -161.652, B 81.275, C -141.67, E1 0, E2 0, E3 0, E4 0}
LIN {X 368.555, Y 208.737, Z 384.548, A -161.652, B 81.275, C -141.67, E1 0, E2 0, E3 0, E4 0}
LIN {X 368.609, Y 208.712, Z 384.542, A -161.652, B 81.275, C -141.67, E1 0, E2 0, E3 0, E4 0}
LIN {X 377.805, Y 164.265, Z 385.35, A -161.652, B 81.275, C -141.67, E1 0, E2 0, E3 0, E4 0}
LIN {X 377.762, Y 163.905, Z 385.373, A -161.652, B 81.275, C -141.67, E1 0, E2 0, E3 0, E4 0}
LIN {X 381.37, Y 147.447, Z 385.643, A -161.652, B 81.275, C -141.67, E1 0, E2 0, E3 0, E4 0}
LIN {X 381.257, Y 147.025, Z 385.68, A -161.652, B 81.275, C -141.67, E1 0, E2 0, E3 0, E4 0}
LIN {X 381.437, Y 146.072, Z 385.7, A -161.652, B 81.275, C -141.67, E1 0, E2 0, E3 0, E4 0}
LIN {X 387.906, Y 144.26, Z 384.845, A -161.652, B 81.275, C -141.67, E1 0, E2 0, E3 0, E4 0}
LIN {X 389.108, Y 144.265, Z 384.669, A -161.652, B 81.275, C -141.67, E1 0, E2 0, E3 0, E4 0}
LIN {X 389.81, Y 144.875, Z 384.538, A -161.652, B 81.275, C -141.67, E1 0, E2 0, E3 0, E4 0}
LIN {X 391.643, Y 149.644, Z 384.04, A -161.652, B 81.275, C -141.67, E1 0, E2 0, E3 0, E4 0}
LIN {X 392.004, Y 150.304, Z 383.956, A -161.652, B 81.275, C -141.67, E1 0, E2 0, E3 0, E4 0}
LIN {X 397.013, Y 167.748, Z 382.383, A -161.652, B 81.275, C -141.67, E1 0, E2 0, E3 0, E4 0}
LIN {X 397.561, Y 168.909, Z 382.247, A -161.652, B 81.275, C -141.67, E1 0, E2 0, E3 0, E4 0}
LIN {X 404.921, Y 196.432, Z 379.845, A -161.652, B 81.275, C -141.67, E1 0, E2 0, E3 0, E4 0}
LIN {X 404.608, Y 196.328, Z 377.697, A -161.652, B 81.275, C -141.67, E1 0, E2 0, E3 0, E4 0}
LIN {X 403.783, Y 191.132, Z 378.068, A -161.652, B 81.275, C -141.67, E1 0, E2 0, E3 0, E4 0}
LIN {X 392.545, Y 152.028, Z 381.594, A -161.652, B 81.275, C -141.67, E1 0, E2 0, E3 0, E4 0}
LIN {X 399.938, Y 198.569, Z 378.269, A -161.652, B 81.275, C -141.67, E1 0, E2 0, E3 0, E4 0}
LIN {X 395.197, Y 200.365, Z 378.873, A -161.652, B 81.275, C -141.67, E1 0, E2 0, E3 0, E4 0}
LIN {X 386.32, Y 144.485, Z 382.866, A -161.652, B 81.275, C -141.67, E1 0, E2 0, E3 0, E4 0}
LIN {X 381.513, Y 145.866, Z 383.499, A -161.652, B 81.275, C -141.67, E1 0, E2 0, E3 0, E4 0}
LIN {X 390.459, Y 202.18, Z 379.475, A -161.652, B 81.275, C -141.67, E1 0, E2 0, E3 0, E4 0}
LIN {X 385.664, Y 203.634, Z 380.104, A -161.652, B 81.275, C -141.67, E1 0, E2 0, E3 0, E4 0}
LIN {X 378.187, Y 156.569, Z 383.466, A -161.652, B 81.275, C -141.67, E1 0, E2 0, E3 0, E4 0}
LIN {X 375.291, Y 169.978, Z 383.241, A -161.652, B 81.275, C -141.67, E1 0, E2 0, E3 0, E4 0}
LIN {X 380.894, Y 205.253, Z 380.72, A -161.652, B 81.275, C -141.67, E1 0, E2 0, E3 0, E4 0}
LIN {X 376.117, Y 206.823, Z 381.34, A -161.652, B 81.275, C -141.67, E1 0, E2 0, E3 0, E4 0}
LIN {X 372.717, Y 185.416, Z 382.87, A -161.652, B 81.275, C -141.67, E1 0, E2 0, E3 0, E4 0}
LIN {X 369.583, Y 197.333, Z 382.75, A -161.652, B 81.275, C -141.67, E1 0, E2 0, E3 0, E4 0}
LIN {X 371.355, Y 208.487, Z 381.953, A -161.652, B 81.275, C -141.67, E1 0, E2 0, E3 0, E4 0}
LIN {X 397.248, Y 168.805, Z 380.099, A -161.652, B 81.275, C -141.67, E1 0, E2 0, E3 0, E4 0}
LIN {X 397.467, Y 169.268, Z 380.044, A -161.652, B 81.275, C -141.67, E1 0, E2 0, E3 0, E4 0}
LIN {X 397.414, Y 169.773, Z 380.028, A -161.652, B 81.275, C -141.67, E1 0, E2 0, E3 0, E4 0}
LIN {X 404.86, Y 193.994, Z 377.773, A -161.652, B 81.275, C -141.67, E1 0, E2 0, E3 0, E4 0}
LIN {X 404.957, Y 195.289, Z 377.696, A -161.652, B 81.275, C -141.67, E1 0, E2 0, E3 0, E4 0}
LIN {X 404.59, Y 196.382, Z 377.697, A -161.652, B 81.275, C -141.67, E1 0, E2 0, E3 0, E4 0}
LIN {X 403.783, Y 197.217, Z 377.774, A -161.652, B 81.275, C -141.67, E1 0, E2 0, E3 0, E4 0}
LIN {X 366.788, Y 209.721, Z 382.559, A -161.652, B 81.275, C -141.67, E1 0, E2 0, E3 0, E4 0}
LIN {X 370.657, Y 192.501, Z 382.827, A -161.652, B 81.275, C -141.67, E1 0, E2 0, E3 0, E4 0}
LIN {X 380.22, Y 146.149, Z 383.674, A -161.652, B 81.275, C -141.67, E1 0, E2 0, E3 0, E4 0}
LIN {X 387.593, Y 144.157, Z 382.696, A -161.652, B 81.275, C -141.67, E1 0, E2 0, E3 0, E4 0}
LIN {X 388.795, Y 144.161, Z 382.521, A -161.652, B 81.275, C -141.67, E1 0, E2 0, E3 0, E4 0}
LIN {X 389.497, Y 144.772, Z 382.389, A -161.652, B 81.275, C -141.67, E1 0, E2 0, E3 0, E4 0}
LIN {X 391.33, Y 149.54, Z 381.892, A -161.652, B 81.275, C -141.67, E1 0, E2 0, E3 0, E4 0}
LIN {X 391.69, Y 150.2, Z 381.807, A -161.652, B 81.275, C -141.67, E1 0, E2 0, E3 0, E4 0}
LIN {X 396.7, Y 167.644, Z 380.235, A -161.652, B 81.275, C -141.67, E1 0, E2 0, E3 0, E4 0}
LIN {X 397.248, Y 168.805, Z 380.099, A -161.652, B 81.275, C -141.67, E1 0, E2 0, E3 0, E4 0}
LIN {X 404.029, Y 191.82, Z 377.999, A -161.652, B 81.275, C -141.67, E1 0, E2 0, E3 0, E4 0}
LIN {X 403.716, Y 191.717, Z 375.85, A -161.652, B 81.275, C -141.67, E1 0, E2 0, E3 0, E4 0}
LIN {X 404.389, Y 195.951, Z 375.548, A -161.652, B 81.275, C -141.67, E1 0, E2 0, E3 0, E4 0}
LIN {X 399.752, Y 198.407, Z 376.104, A -161.652, B 81.275, C -141.67, E1 0, E2 0, E3 0, E4 0}
LIN {X 392.463, Y 152.522, Z 379.383, A -161.652, B 81.275, C -141.67, E1 0, E2 0, E3 0, E4 0}
LIN {X 386.139, Y 144.354, Z 380.699, A -161.652, B 81.275, C -141.67, E1 0, E2 0, E3 0, E4 0}
LIN {X 395.013, Y 200.214, Z 376.707, A -161.652, B 81.275, C -141.67, E1 0, E2 0, E3 0, E4 0}
LIN {X 390.276, Y 202.034, Z 377.31, A -161.652, B 81.275, C -141.67, E1 0, E2 0, E3 0, E4 0}
LIN {X 381.329, Y 145.716, Z 381.334, A -161.652, B 81.275, C -141.67, E1 0, E2 0, E3 0, E4 0}
LIN {X 377.724, Y 154.661, Z 381.427, A -161.652, B 81.275, C -141.67, E1 0, E2 0, E3 0, E4 0}
LIN {X 385.479, Y 203.482, Z 377.938, A -161.652, B 81.275, C -141.67, E1 0, E2 0, E3 0, E4 0}
LIN {X 380.711, Y 205.104, Z 378.555, A -161.652, B 81.275, C -141.67, E1 0, E2 0, E3 0, E4 0}
LIN {X 374.894, Y 168.485, Z 381.171, A -161.652, B 81.275, C -141.67, E1 0, E2 0, E3 0, E4 0}
LIN {X 372.001, Y 181.918, Z 380.943, A -161.652, B 81.275, C -141.67, E1 0, E2 0, E3 0, E4 0}
LIN {X 375.934, Y 206.673, Z 379.175, A -161.652, B 81.275, C -141.67, E1 0, E2 0, E3 0, E4 0}
LIN {X 371.172, Y 208.339, Z 379.788, A -161.652, B 81.275, C -141.67, E1 0, E2 0, E3 0, E4 0}
LIN {X 369.121, Y 195.428, Z 380.711, A -161.652, B 81.275, C -141.67, E1 0, E2 0, E3 0, E4 0}
LIN {X 366.122, Y 208.193, Z 380.53, A -161.652, B 81.275, C -141.67, E1 0, E2 0, E3 0, E4 0}
LIN {X 366.356, Y 209.664, Z 380.425, A -161.652, B 81.275, C -141.67, E1 0, E2 0, E3 0, E4 0}
LIN {X 396.935, Y 168.702, Z 377.95, A -161.652, B 81.275, C -141.67, E1 0, E2 0, E3 0, E4 0}
LIN {X 397.154, Y 169.165, Z 377.896, A -161.652, B 81.275, C -141.67, E1 0, E2 0, E3 0, E4 0}
LIN {X 397.101, Y 169.669, Z 377.879, A -161.652, B 81.275, C -141.67, E1 0, E2 0, E3 0, E4 0}
LIN {X 404.547, Y 193.89, Z 375.624, A -161.652, B 81.275, C -141.67, E1 0, E2 0, E3 0, E4 0}
LIN {X 404.644, Y 195.185, Z 375.548, A -161.652, B 81.275, C -141.67, E1 0, E2 0, E3 0, E4 0}
LIN {X 404.277, Y 196.279, Z 375.548, A -161.652, B 81.275, C -141.67, E1 0, E2 0, E3 0, E4 0}
LIN {X 403.47, Y 197.113, Z 375.625, A -161.652, B 81.275, C -141.67, E1 0, E2 0, E3 0, E4 0}
LIN {X 367.412, Y 209.283, Z 380.29, A -161.652, B 81.275, C -141.67, E1 0, E2 0, E3 0, E4 0}
LIN {X 365.679, Y 209.931, Z 380.511, A -161.652, B 81.275, C -141.67, E1 0, E2 0, E3 0, E4 0}
LIN {X 377.876, Y 153.987, Z 381.437, A -161.652, B 81.275, C -141.67, E1 0, E2 0, E3 0, E4 0}
LIN {X 377.952, Y 153.908, Z 381.43, A -161.652, B 81.275, C -141.67, E1 0, E2 0, E3 0, E4 0}
LIN {X 379.218, Y 146.367, Z 381.61, A -161.652, B 81.275, C -141.67, E1 0, E2 0, E3 0, E4 0}
LIN {X 387.28, Y 144.053, Z 380.547, A -161.652, B 81.275, C -141.67, E1 0, E2 0, E3 0, E4 0}
LIN {X 388.482, Y 144.058, Z 380.372, A -161.652, B 81.275, C -141.67, E1 0, E2 0, E3 0, E4 0}
LIN {X 389.184, Y 144.668, Z 380.24, A -161.652, B 81.275, C -141.67, E1 0, E2 0, E3 0, E4 0}
LIN {X 391.017, Y 149.436, Z 379.743, A -161.652, B 81.275, C -141.67, E1 0, E2 0, E3 0, E4 0}
LIN {X 391.377, Y 150.096, Z 379.658, A -161.652, B 81.275, C -141.67, E1 0, E2 0, E3 0, E4 0}
LIN {X 396.387, Y 167.54, Z 378.086, A -161.652, B 81.275, C -141.67, E1 0, E2 0, E3 0, E4 0}
LIN {X 396.935, Y 168.702, Z 377.95, A -161.652, B 81.275, C -141.67, E1 0, E2 0, E3 0, E4 0}
PTP {X 400.878, Y 198.448, Z 421.334, A -161.652, B 81.275, C -141.67, E1 0, E2 0, E3 0, E4 0, S 'B010'}
PTP {A1 5, A2 -90, A3 100, A4 5, A5 -10, A6 -5, E1 0, E2 0, E3 0, E4 0} C_PTP

END
